(*

short summary
==================
This class tests all methods of LDT assertions
with various combinations of inputs and checks expected 
outputs are satisfied or not

.. <legal notes>

legal notes
=================
| SPDX-FileCopyrightText: © 2022 ekvip automation GmbH <info@ekvip.de>
| SPDX-License-Identifier: Apache-2.0
| For details check: Apache-2.0_

.. _Apache-2.0: https://www.apache.org/licenses/LICENSE-2.0

.. </legal notes>

methods and properties
======================

*)


FUNCTION_BLOCK LDTAssertionTests EXTENDS AbstractAssertorTest
VAR
	
END_VAR
VAR CONSTANT
	(* prefix to unify the test names *)
	TEST_NAME_PREFIX		:STRING := 'assert.dateAndTime.long.dateAndTime.';
	(* max value of a LWORD *)
	{attribute 'hide'}
	MAX_LWORD				:LWORD := 16#FFFF_FFFF_FFFF_FFFF;
	(* min value of a LWORD *)
	{attribute 'hide'}
	MIN_LWORD				:LWORD := 16#0000_0000_0000_0000;
	(* only the msb is set *)
	{attribute 'hide'}
	MSB_ONLY				:LWORD := 16#8000_0000_0000_0000;
	(* only the msb is set *)
	{attribute 'hide'}
	LSB_ONLY				:LWORD := 16#0000_0000_0000_0001;
	(* all bits set except the msb *)
	{attribute 'hide'}
	WITHOUT_MSB 			:LWORD := 16#7FFF_FFFF_FFFF_FFFF;
	(* for every nibble is the msb set only *)
	{attribute 'hide'}
	ALL_NIBBLE_MSB			:LWORD := 16#8888_8888_8888_8888;
	(* for every nibble is the msb unset only *)
	{attribute 'hide'}
	WITHOUT_NIBBLE_MSB		:LWORD := 16#7777_7777_7777_7777;
	(* for every nibble is the lsb set only *)
	{attribute 'hide'}
	ALL_NIBBLE_LSB			:LWORD := 16#1111_1111_1111_1111;
	(* every bit is set except the lsb *)
	{attribute 'hide'}
	LSB_IS_UNSET			:LWORD := 16#FFFF__FFFF_FFFF_FFFE;
	(* max vale of date and time *)
	LDT_MAX					:LDT := TO_LDT(MAX_LWORD);
	(* min vale of date and time *)
	LDT_MIN					:LDT := TO_LDT(MIN_LWORD);
	(* only the msb is set *)
	LDT_MSB_ONLY			:LDT := TO_LDT(MSB_ONLY);
	(* all bits set except the msb *)
	LDT_WITHOUT_MSB 		:LDT := TO_LDT(WITHOUT_MSB);
	(* for every nibble is the msb set only *)
	LDT_ALL_NIBBLE_MSB		:LDT := TO_LDT(ALL_NIBBLE_MSB);
	(* for every nibble is the msb unset only *)
	LDT_WITHOUT_NIBBLE_MSB	:LDT := TO_LDT(WITHOUT_NIBBLE_MSB);
	(* for every nibble is the lsb set only *)
	LDT_ALL_NIBBLE_LSB		:LDT := TO_LDT(ALL_NIBBLE_LSB);	
	(* every bit is set except the lsb *)
	LDT_LSB_IS_UNSET		:LDT := TO_LDT(LSB_IS_UNSET);
	(* only the msb is set *)
	LDT_LSB_ONLY			:LDT := TO_LDT(LSB_ONLY);
END_VAR

THIS^.runValueIsEqualToTests();
THIS^.runValueIsGreaterThanTests();
THIS^.runValueIsInRangeOfTests();
THIS^.runValueIsLessThanTests();
THIS^.runValueIsMaxTests();
THIS^.runValueIsMinTests();
THIS^.runValueIsNotEqualToTests();

(*

short summary
==================
This test method is a helper function to create a unified test name

.. <legal notes>

legal notes
=================
| SPDX-FileCopyrightText: © 2022 ekvip automation GmbH <info@ekvip.de>
| SPDX-License-Identifier: Apache-2.0
| For details check: Apache-2.0_

.. _Apache-2.0: https://www.apache.org/licenses/LICENSE-2.0

.. </legal notes>

parameters
==========

*)

METHOD PROTECTED getTestNameFor :Tc2_System.T_MaxString
VAR_INPUT
	(* name of the method to test, to create a unified test name *)
	nameOfMethodToTest	:Tc2_System.T_MaxString;
END_VAR
getTestNameFor := Tc2_Standard.CONCAT(THIS^.TEST_NAME_PREFIX, nameOfMethodToTest);
END_METHOD

(*

short summary
==================
This test method tests ``assert.dateAndTime.long.dateAndTime.valueIsEqualTo``
method of CNM_AssertionInterfaces library with various inputs

.. <legal notes>

legal notes
=================
| SPDX-FileCopyrightText: © 2022 ekvip automation GmbH <info@ekvip.de>
| SPDX-License-Identifier: Apache-2.0
| For details check: Apache-2.0_

.. _Apache-2.0: https://www.apache.org/licenses/LICENSE-2.0

.. </legal notes>

*)

METHOD runValueIsEqualToTests
RETURN (NOT TcUnit.TEST_ORDERED(THIS^.getTestNameFor('valueIsEqualTo')));

THIS^.testValueIsEqualTo(
	valueToTest := THIS^.LDT_MAX,
	expected := THIS^.LDT_MAX
);
THIS^.testValueIsEqualTo(
	valueToTest := THIS^.LDT_MIN,
	expected := THIS^.LDT_MIN
);
THIS^.testValueIsEqualTo(
	valueToTest := THIS^.LDT_MIN,
	expected := THIS^.LDT_MAX
);
THIS^.testValueIsEqualTo(
	valueToTest := THIS^.LDT_MAX,
	expected := THIS^.LDT_MIN
);
THIS^.testValueIsEqualTo(
	valueToTest := THIS^.LDT_ALL_NIBBLE_LSB,
	expected := THIS^.LDT_ALL_NIBBLE_LSB
);
THIS^.testValueIsEqualTo(
	valueToTest := THIS^.LDT_LSB_ONLY,
	expected := THIS^.LDT_MSB_ONLY
);
THIS^.testValueIsEqualTo(
	valueToTest := THIS^.LDT_MSB_ONLY,
	expected := THIS^.LDT_MSB_ONLY
);
THIS^.testValueIsEqualTo(
	valueToTest := THIS^.LDT_MSB_ONLY,
	expected := THIS^.LDT_LSB_ONLY
);

TcUnit.TEST_FINISHED();
END_METHOD

(*

short summary
==================
This test method tests ``assert.dateAndTime.long.dateAndTime.valueIsGreaterThan``
method of CNM_AssertionInterfaces library with various inputs

.. <legal notes>

legal notes
=================
| SPDX-FileCopyrightText: © 2022 ekvip automation GmbH <info@ekvip.de>
| SPDX-License-Identifier: Apache-2.0
| For details check: Apache-2.0_

.. _Apache-2.0: https://www.apache.org/licenses/LICENSE-2.0

.. </legal notes>

*)

METHOD runValueIsGreaterThanTests
RETURN (NOT TcUnit.TEST_ORDERED(THIS^.getTestNameFor('valueIsGreaterThan')));

THIS^.testValueIsGreaterThan(
	valueToTest := THIS^.LDT_MAX,
	lessValue := THIS^.LDT_MAX
);
THIS^.testValueIsGreaterThan(
	valueToTest := THIS^.LDT_MIN,
	lessValue := THIS^.LDT_MIN
);
THIS^.testValueIsGreaterThan(
	valueToTest := THIS^.LDT_MIN,
	lessValue := THIS^.LDT_MAX
);
THIS^.testValueIsGreaterThan(
	valueToTest := THIS^.LDT_MAX,
	lessValue := THIS^.LDT_MIN
);
THIS^.testValueIsGreaterThan(
	valueToTest := THIS^.LDT_ALL_NIBBLE_LSB,
	lessValue := THIS^.LDT_ALL_NIBBLE_LSB
);
THIS^.testValueIsGreaterThan(
	valueToTest := THIS^.LDT_ALL_NIBBLE_MSB,
	lessValue := THIS^.LDT_ALL_NIBBLE_LSB
);
THIS^.testValueIsGreaterThan(
	valueToTest := THIS^.LDT_ALL_NIBBLE_LSB,
	lessValue := THIS^.LDT_ALL_NIBBLE_MSB
);
THIS^.testValueIsGreaterThan(
	valueToTest := THIS^.LDT_LSB_ONLY,
	lessValue := THIS^.LDT_MSB_ONLY
);
THIS^.testValueIsGreaterThan(
	valueToTest := THIS^.LDT_MSB_ONLY,
	lessValue := THIS^.LDT_MSB_ONLY
);
THIS^.testValueIsGreaterThan(
	valueToTest := THIS^.LDT_MSB_ONLY,
	lessValue := THIS^.LDT_LSB_ONLY
);
THIS^.testValueIsGreaterThan(
	valueToTest := THIS^.LDT_LSB_IS_UNSET,
	lessValue := THIS^.LDT_MAX
);
THIS^.testValueIsGreaterThan(
	valueToTest := THIS^.LDT_MAX,
	lessValue := THIS^.LDT_LSB_IS_UNSET
);

TcUnit.TEST_FINISHED();
END_METHOD

(*

short summary
==================
This test method tests ``assert.dateAndTime.long.dateAndTime.valueIsInRangeOf``
method of CNM_AssertionInterfaces library with various inputs

.. <legal notes>

legal notes
=================
| SPDX-FileCopyrightText: © 2022 ekvip automation GmbH <info@ekvip.de>
| SPDX-License-Identifier: Apache-2.0
| For details check: Apache-2.0_

.. _Apache-2.0: https://www.apache.org/licenses/LICENSE-2.0

.. </legal notes>

*)

METHOD runValueIsInRangeOfTests
RETURN (NOT TcUnit.TEST_ORDERED(THIS^.getTestNameFor('valueIsInRangeOf')));

THIS^.testValueIsInRangeOf(
	lowerLimit := THIS^.LDT_MIN,
	valueToTest := THIS^.LDT_MAX,
	upperLimit	:= THIS^.LDT_MAX
);
THIS^.testValueIsInRangeOf(
	lowerLimit := THIS^.LDT_MIN,
	valueToTest := THIS^.LDT_MIN,
	upperLimit	:= THIS^.LDT_MAX
);
THIS^.testValueIsInRangeOf(
	lowerLimit := THIS^.LDT_MAX,
	valueToTest := THIS^.LDT_MAX,
	upperLimit	:= THIS^.LDT_MIN
);
THIS^.testValueIsInRangeOf(
	lowerLimit := THIS^.LDT_MAX,
	valueToTest := THIS^.LDT_MIN,
	upperLimit	:= THIS^.LDT_MIN
);
THIS^.testValueIsInRangeOf(
	lowerLimit := THIS^.LDT_LSB_IS_UNSET,
	valueToTest := THIS^.LDT_MIN,
	upperLimit	:= THIS^.LDT_MAX
);
THIS^.testValueIsInRangeOf(
	lowerLimit := THIS^.LDT_MIN,
	valueToTest := THIS^.LDT_LSB_IS_UNSET,
	upperLimit	:= THIS^.LDT_MAX
);
THIS^.testValueIsInRangeOf(
	lowerLimit := THIS^.LDT_LSB_IS_UNSET,
	valueToTest := THIS^.LDT_LSB_IS_UNSET,
	upperLimit	:= THIS^.LDT_LSB_IS_UNSET
);
THIS^.testValueIsInRangeOf(
	lowerLimit := THIS^.LDT_ALL_NIBBLE_LSB,
	valueToTest := THIS^.LDT_LSB_IS_UNSET,
	upperLimit	:= THIS^.LDT_ALL_NIBBLE_MSB
);
THIS^.testValueIsInRangeOf(
	lowerLimit := THIS^.LDT_LSB_IS_UNSET,
	valueToTest := THIS^.LDT_ALL_NIBBLE_LSB,
	upperLimit	:= THIS^.LDT_ALL_NIBBLE_MSB
);
THIS^.testValueIsInRangeOf(
	lowerLimit := THIS^.LDT_LSB_ONLY,
	valueToTest := THIS^.LDT_WITHOUT_MSB,
	upperLimit	:= THIS^.LDT_MSB_ONLY
);
THIS^.testValueIsInRangeOf(
	lowerLimit := THIS^.LDT_WITHOUT_MSB,
	valueToTest := THIS^.LDT_LSB_ONLY,
	upperLimit	:= THIS^.LDT_MSB_ONLY
);
THIS^.testValueIsInRangeOf(
	lowerLimit := THIS^.LDT_WITHOUT_NIBBLE_MSB,
	valueToTest := THIS^.LDT_MAX,
	upperLimit	:= THIS^.LDT_ALL_NIBBLE_MSB
);
THIS^.testValueIsInRangeOf(
	lowerLimit := THIS^.LDT_WITHOUT_NIBBLE_MSB,
	valueToTest := THIS^.LDT_MIN,
	upperLimit	:= THIS^.LDT_ALL_NIBBLE_MSB
);
THIS^.testValueIsInRangeOf(
	lowerLimit := THIS^.LDT_WITHOUT_NIBBLE_MSB,
	valueToTest := THIS^.LDT_WITHOUT_NIBBLE_MSB,
	upperLimit	:= THIS^.LDT_ALL_NIBBLE_MSB
);
THIS^.testValueIsInRangeOf(
	lowerLimit := THIS^.LDT_WITHOUT_NIBBLE_MSB,
	valueToTest := THIS^.LDT_ALL_NIBBLE_MSB,
	upperLimit	:= THIS^.LDT_ALL_NIBBLE_MSB
);

TcUnit.TEST_FINISHED();
END_METHOD

(*

short summary
==================
This test method tests ``assert.dateAndTime.long.dateAndTime.valueIsLessThan``
method of CNM_AssertionInterfaces library with various inputs

.. <legal notes>

legal notes
=================
| SPDX-FileCopyrightText: © 2022 ekvip automation GmbH <info@ekvip.de>
| SPDX-License-Identifier: Apache-2.0
| For details check: Apache-2.0_

.. _Apache-2.0: https://www.apache.org/licenses/LICENSE-2.0

.. </legal notes>

*)

METHOD runValueIsLessThanTests
RETURN (NOT TcUnit.TEST_ORDERED(THIS^.getTestNameFor('valueIsLessThan')));

THIS^.testValueIsLessThan(
	valueToTest := THIS^.LDT_MAX,
	greaterValue := THIS^.LDT_MAX
);
THIS^.testValueIsLessThan(
	valueToTest := THIS^.LDT_MIN,
	greaterValue := THIS^.LDT_MIN
);
THIS^.testValueIsLessThan(
	valueToTest := THIS^.LDT_MIN,
	greaterValue := THIS^.LDT_MAX
);
THIS^.testValueIsLessThan(
	valueToTest := THIS^.LDT_MAX,
	greaterValue := THIS^.LDT_MIN
);
THIS^.testValueIsLessThan(
	valueToTest := THIS^.LDT_ALL_NIBBLE_LSB,
	greaterValue := THIS^.LDT_ALL_NIBBLE_LSB
);
THIS^.testValueIsLessThan(
	valueToTest := THIS^.LDT_ALL_NIBBLE_MSB,
	greaterValue := THIS^.LDT_ALL_NIBBLE_LSB
);
THIS^.testValueIsLessThan(
	valueToTest := THIS^.LDT_ALL_NIBBLE_LSB,
	greaterValue := THIS^.LDT_ALL_NIBBLE_MSB
);
THIS^.testValueIsLessThan(
	valueToTest := THIS^.LDT_LSB_ONLY,
	greaterValue := THIS^.LDT_MSB_ONLY
);
THIS^.testValueIsLessThan(
	valueToTest := THIS^.LDT_MSB_ONLY,
	greaterValue := THIS^.LDT_MSB_ONLY
);
THIS^.testValueIsLessThan(
	valueToTest := THIS^.LDT_MSB_ONLY,
	greaterValue := THIS^.LDT_LSB_ONLY
);
THIS^.testValueIsLessThan(
	valueToTest := THIS^.LDT_LSB_IS_UNSET,
	greaterValue := THIS^.LDT_MAX
);
THIS^.testValueIsLessThan(
	valueToTest := THIS^.LDT_MAX,
	greaterValue := THIS^.LDT_LSB_IS_UNSET
);

TcUnit.TEST_FINISHED();
END_METHOD

(*

short summary
==================
This test method tests ``assert.dateAndTime.long.dateAndTime.valueIsMax``
method of CNM_AssertionInterfaces library with various inputs

.. <legal notes>

legal notes
=================
| SPDX-FileCopyrightText: © 2022 ekvip automation GmbH <info@ekvip.de>
| SPDX-License-Identifier: Apache-2.0
| For details check: Apache-2.0_

.. _Apache-2.0: https://www.apache.org/licenses/LICENSE-2.0

.. </legal notes>

*)

METHOD runValueIsMaxTests
RETURN (NOT TcUnit.TEST_ORDERED(THIS^.getTestNameFor('valueIsMax')));

THIS^.testValueIsMax(
	valueToTest := THIS^.LDT_MAX,
	maximumValue := THIS^.LDT_MAX
);
THIS^.testValueIsMax(
	valueToTest := THIS^.LDT_MIN,
	maximumValue := THIS^.LDT_MIN
);
THIS^.testValueIsMax(
	valueToTest := THIS^.LDT_MIN,
	maximumValue := THIS^.LDT_MAX
);
THIS^.testValueIsMax(
	valueToTest := THIS^.LDT_MAX,
	maximumValue := THIS^.LDT_MIN
);
THIS^.testValueIsMax(
	valueToTest := THIS^.LDT_ALL_NIBBLE_LSB,
	maximumValue := THIS^.LDT_ALL_NIBBLE_LSB
);
THIS^.testValueIsMax(
	valueToTest := THIS^.LDT_ALL_NIBBLE_MSB,
	maximumValue := THIS^.LDT_ALL_NIBBLE_LSB
);
THIS^.testValueIsMax(
	valueToTest := THIS^.LDT_ALL_NIBBLE_LSB,
	maximumValue := THIS^.LDT_ALL_NIBBLE_MSB
);
THIS^.testValueIsMax(
	valueToTest := THIS^.LDT_LSB_ONLY,
	maximumValue := THIS^.LDT_MSB_ONLY
);
THIS^.testValueIsMax(
	valueToTest := THIS^.LDT_MSB_ONLY,
	maximumValue := THIS^.LDT_MSB_ONLY
);
THIS^.testValueIsMax(
	valueToTest := THIS^.LDT_MSB_ONLY,
	maximumValue := THIS^.LDT_LSB_ONLY
);
THIS^.testValueIsMax(
	valueToTest := THIS^.LDT_LSB_IS_UNSET,
	maximumValue := THIS^.LDT_MAX
);
THIS^.testValueIsMax(
	valueToTest := THIS^.LDT_MAX,
	maximumValue := THIS^.LDT_LSB_IS_UNSET
);

TcUnit.TEST_FINISHED();
END_METHOD

(*

short summary
==================
This test method tests ``assert.dateAndTime.long.dateAndTime.valueIsMin``
method of CNM_AssertionInterfaces library with various inputs

.. <legal notes>

legal notes
=================
| SPDX-FileCopyrightText: © 2022 ekvip automation GmbH <info@ekvip.de>
| SPDX-License-Identifier: Apache-2.0
| For details check: Apache-2.0_

.. _Apache-2.0: https://www.apache.org/licenses/LICENSE-2.0

.. </legal notes>

*)

METHOD runValueIsMinTests
RETURN (NOT TcUnit.TEST_ORDERED(THIS^.getTestNameFor('valueIsMin')));

THIS^.testValueIsMin(
	valueToTest := THIS^.LDT_MAX,
	minimumValue := THIS^.LDT_MAX
);
THIS^.testValueIsMin(
	valueToTest := THIS^.LDT_MIN,
	minimumValue := THIS^.LDT_MIN
);
THIS^.testValueIsMin(
	valueToTest := THIS^.LDT_MIN,
	minimumValue := THIS^.LDT_MAX
);
THIS^.testValueIsMin(
	valueToTest := THIS^.LDT_MAX,
	minimumValue := THIS^.LDT_MIN
);
THIS^.testValueIsMin(
	valueToTest := THIS^.LDT_ALL_NIBBLE_LSB,
	minimumValue := THIS^.LDT_ALL_NIBBLE_LSB
);
THIS^.testValueIsMin(
	valueToTest := THIS^.LDT_ALL_NIBBLE_MSB,
	minimumValue := THIS^.LDT_ALL_NIBBLE_LSB
);
THIS^.testValueIsMin(
	valueToTest := THIS^.LDT_ALL_NIBBLE_LSB,
	minimumValue := THIS^.LDT_ALL_NIBBLE_MSB
);
THIS^.testValueIsMin(
	valueToTest := THIS^.LDT_LSB_ONLY,
	minimumValue := THIS^.LDT_MSB_ONLY
);
THIS^.testValueIsMin(
	valueToTest := THIS^.LDT_MSB_ONLY,
	minimumValue := THIS^.LDT_MSB_ONLY
);
THIS^.testValueIsMin(
	valueToTest := THIS^.LDT_MSB_ONLY,
	minimumValue := THIS^.LDT_LSB_ONLY
);
THIS^.testValueIsMin(
	valueToTest := THIS^.LDT_LSB_IS_UNSET,
	minimumValue := THIS^.LDT_MAX
);
THIS^.testValueIsMin(
	valueToTest := THIS^.LDT_MAX,
	minimumValue := THIS^.LDT_LSB_IS_UNSET
);

TcUnit.TEST_FINISHED();
END_METHOD

(*

short summary
==================
This test method tests ``assert.dateAndTime.long.dateAndTime.valueIsNotEqualTo``
method of CNM_AssertionInterfaces library with various inputs

.. <legal notes>

legal notes
=================
| SPDX-FileCopyrightText: © 2022 ekvip automation GmbH <info@ekvip.de>
| SPDX-License-Identifier: Apache-2.0
| For details check: Apache-2.0_

.. _Apache-2.0: https://www.apache.org/licenses/LICENSE-2.0

.. </legal notes>

*)

METHOD runValueIsNotEqualToTests
RETURN (NOT TcUnit.TEST_ORDERED(THIS^.getTestNameFor('valueIsNotEqualTo')));

THIS^.testValueIsNotEqualTo(
	valueToTest := THIS^.LDT_MAX,
	unexpectedValue := THIS^.LDT_MAX
);
THIS^.testValueIsNotEqualTo(
	valueToTest := THIS^.LDT_MIN,
	unexpectedValue := THIS^.LDT_MIN
);
THIS^.testValueIsNotEqualTo(
	valueToTest := THIS^.LDT_MIN,
	unexpectedValue := THIS^.LDT_MAX
);
THIS^.testValueIsNotEqualTo(
	valueToTest := THIS^.LDT_MAX,
	unexpectedValue := THIS^.LDT_MIN
);
THIS^.testValueIsNotEqualTo(
	valueToTest := THIS^.LDT_ALL_NIBBLE_LSB,
	unexpectedValue := THIS^.LDT_ALL_NIBBLE_LSB
);
THIS^.testValueIsNotEqualTo(
	valueToTest := THIS^.LDT_LSB_ONLY,
	unexpectedValue := THIS^.LDT_MSB_ONLY
);
THIS^.testValueIsNotEqualTo(
	valueToTest := THIS^.LDT_MSB_ONLY,
	unexpectedValue := THIS^.LDT_MSB_ONLY
);
THIS^.testValueIsNotEqualTo(
	valueToTest := THIS^.LDT_MSB_ONLY,
	unexpectedValue := THIS^.LDT_LSB_ONLY
);

TcUnit.TEST_FINISHED();
END_METHOD

(*

short summary
==================
This test method tests ``assert.dateAndTime.long.dateAndTime.valueIsEqualTo``
method of CNM_AssertionInterfaces library, 
it provides the possibility to handover test data via parameter 


.. <legal notes>

legal notes
=================
| SPDX-FileCopyrightText: © 2022 ekvip automation GmbH <info@ekvip.de>
| SPDX-License-Identifier: Apache-2.0
| For details check: Apache-2.0_

.. _Apache-2.0: https://www.apache.org/licenses/LICENSE-2.0

.. </legal notes>

parameters
==========

*)

METHOD testValueIsEqualTo 
VAR_INPUT
	(* for the test it's the parameter ``currentValue`` *)
	valueToTest	:LDT;
	(* for the test it's the parameter ``expectedValue`` *)
	expected	:LDT;
END_VAR
VAR
	(* just the expectation if the assertion to test must be worng or true *)
	assertionIsWrong		:BOOL;
	(* contains the format string for the test message *)
	message					:Tc2_System.T_MaxString;
	(* TwinCAT printf with the test message *)
	messageStringBuilder	:Tc2_Utilities.FB_FormatString;
	(* LDT value of ``currentValue`` as string *)
	currentValueAsString	:STRING(22);
	(* LDT value of ``expectedValue`` as string *)
	expectedValueAsString	:STRING(22);
END_VAR
THIS^.assertorContainer.resetAssertor();

assertionIsWrong := (valueToTest <> expected);

message := SEL(
	assertionIsWrong,
	'currentValue is %s expectedValue is %s assertion must be TRUE', 
	'currentValue is %s expectedValue is %s assertion must be FALSE'
);
currentValueAsString := TO_STRING(valueToTest);
expectedValueAsString := TO_STRING(expected);

messageStringBuilder(
	sFormat := message,
	arg1 := THIS^.AnyToArg(currentValueAsString),
	arg2 := THIS^.AnyToArg(expectedValueAsString)
);

THIS^.assertorContainer.assertor.assert.dateAndTime.long.dateAndTime.valueIsEqualTo(
	currentValue	:= valueToTest,
	expectedValue	:= expected,
	message			:= ''
);

THIS^.AssertEquals_BOOL(
	Expected 	:= assertionIsWrong,
	Actual 		:= THIS^.assertorContainer.wasAssertionWrong,
	Message 	:= messageStringBuilder.sOut
);
END_METHOD

(*

short summary
==================
This test method tests ``assert.dateAndTime.long.dateAndTime.valueIsGreaterThan``
method of CNM_AssertionInterfaces library, 
it provides the possibility to handover test data via parameter 


.. <legal notes>

legal notes
=================
| SPDX-FileCopyrightText: © 2022 ekvip automation GmbH <info@ekvip.de>
| SPDX-License-Identifier: Apache-2.0
| For details check: Apache-2.0_

.. _Apache-2.0: https://www.apache.org/licenses/LICENSE-2.0

.. </legal notes>

parameters
==========

*)

METHOD testValueIsGreaterThan 
VAR_INPUT
	(* for the test it's the parameter ``currentValue`` *)
	valueToTest	:LDT;
	(* for the test it's the parameter ``lessValue`` *)
	lessValue	:LDT;
END_VAR
VAR
	(* just the expectation if the assertion to test must be worng or true *)
	assertionIsWrong		:BOOL;
	(* contains the format string for the test message *)
	message					:Tc2_System.T_MaxString;
	(* TwinCAT printf with the test message *)
	messageStringBuilder	:Tc2_Utilities.FB_FormatString;
	(* LDT value of ``currentValue`` as string *)
	currentValueAsString	:STRING(22);
	(* LDT value of ``lessValue`` as string *)
	lessValueAsString		:STRING(22);
END_VAR
THIS^.assertorContainer.resetAssertor();

assertionIsWrong := (valueToTest <= lessValue);

message := SEL(
	assertionIsWrong,
	'currentValue is %s lessValue is %s assertion must be TRUE', 
	'currentValue is %s lessValue is %s assertion must be FALSE'
);
currentValueAsString := TO_STRING(valueToTest);
lessValueAsString := TO_STRING(lessValue);

messageStringBuilder(
	sFormat := message,
	arg1 := THIS^.AnyToArg(currentValueAsString),
	arg2 := THIS^.AnyToArg(lessValueAsString)
);

THIS^.assertorContainer.assertor.assert.dateAndTime.long.dateAndTime.valueIsGreaterThan(
	currentValue	:= valueToTest,
	lessValue		:= lessValue,
	message			:= ''
);

THIS^.AssertEquals_BOOL(
	Expected 	:= assertionIsWrong,
	Actual 		:= THIS^.assertorContainer.wasAssertionWrong,
	Message 	:= messageStringBuilder.sOut
);
END_METHOD

(*

short summary
==================
This test method tests ``assert.dateAndTime.long.dateAndTime.valueIsInRangeOf``
method of CNM_AssertionInterfaces library, 
it provides the possibility to handover test data via parameter 


.. <legal notes>

legal notes
=================
| SPDX-FileCopyrightText: © 2022 ekvip automation GmbH <info@ekvip.de>
| SPDX-License-Identifier: Apache-2.0
| For details check: Apache-2.0_

.. _Apache-2.0: https://www.apache.org/licenses/LICENSE-2.0

.. </legal notes>

parameters
==========

*)

METHOD testValueIsInRangeOf 
VAR_INPUT
	(* for the test it's the parameter ``lowerLimit`` *)
	lowerLimit	:LDT;
	(* for the test it's the parameter ``currentValue`` *)
	valueToTest	:LDT;
	(* for the test it's the parameter ``upperLimit`` *)
	upperLimit	:LDT;
END_VAR
VAR
	(* just the expectation if the assertion to test must be worng or true *)
	assertionIsWrong		:BOOL;
	(* contains the format string for the test message *)
	message					:Tc2_System.T_MaxString;
	(* TwinCAT printf with the test message *)
	messageStringBuilder	:Tc2_Utilities.FB_FormatString;
	(* LDT value of ``lowerLimit`` as string *)
	lowerLimitAsString		:STRING(22);
	(* LDT value of ``currentValue`` as string *)
	currentValueAsString	:STRING(22);
	(* dt value of ``upperLimit`` as string *)
	upperLimitAsString		:STRING(22);

END_VAR
THIS^.assertorContainer.resetAssertor();

assertionIsWrong := ((
		valueToTest < lowerLimit
	) OR (
		valueToTest > upperLimit
	)
);

message := SEL(
	assertionIsWrong,
	'lowerLimit is %s currentValue is %s upperLimit is %s assertion must be TRUE', 
	'lowerLimit is %s currentValue is %s upperLimit is %s assertion must be FALSE'
);
lowerLimitAsString		:= TO_STRING(lowerLimit);
currentValueAsString	:= TO_STRING(valueToTest);
upperLimitAsString		:= TO_STRING(upperLimit);

messageStringBuilder(
	sFormat := message,
	arg1 := THIS^.AnyToArg(lowerLimitAsString),
	arg2 := THIS^.AnyToArg(currentValueAsString),
	arg3 := THIS^.AnyToArg(upperLimitAsString)
);

THIS^.assertorContainer.assertor.assert.dateAndTime.long.dateAndTime.valueIsInRangeOf(
	lowerLimit		:= lowerLimit,
	currentValue	:= valueToTest,
	upperLimit		:= upperLimit,
	message			:= ''
);

THIS^.AssertEquals_BOOL(
	Expected 	:= assertionIsWrong,
	Actual 		:= THIS^.assertorContainer.wasAssertionWrong,
	Message 	:= messageStringBuilder.sOut
);
END_METHOD

(*

short summary
==================
This test method tests ``assert.dateAndTime.long.dateAndTime.valueIsLessThan``
method of CNM_AssertionInterfaces library, 
it provides the possibility to handover test data via parameter 


.. <legal notes>

legal notes
=================
| SPDX-FileCopyrightText: © 2022 ekvip automation GmbH <info@ekvip.de>
| SPDX-License-Identifier: Apache-2.0
| For details check: Apache-2.0_

.. _Apache-2.0: https://www.apache.org/licenses/LICENSE-2.0

.. </legal notes>

parameters
==========

*)

METHOD testValueIsLessThan 
VAR_INPUT
	(* for the test it's the parameter ``currentValue`` *)
	valueToTest		:LDT;
	(* for the test it's the parameter ``greaterValue`` *)
	greaterValue	:LDT;
END_VAR
VAR
	(* just the expectation if the assertion to test must be worng or true *)
	assertionIsWrong		:BOOL;
	(* contains the format string for the test message *)
	message					:Tc2_System.T_MaxString;
	(* TwinCAT printf with the test message *)
	messageStringBuilder	:Tc2_Utilities.FB_FormatString;
	(* LDT value of ``currentValue`` as string *)
	currentValueAsString	:STRING(22);
	(* LDT value of ``greaterValue`` as string *)
	greaterValueAsString	:STRING(22);
END_VAR
THIS^.assertorContainer.resetAssertor();

assertionIsWrong := (valueToTest >= greaterValue);

message := SEL(
	assertionIsWrong,
	'currentValue is %s greaterValue is %s assertion must be TRUE', 
	'currentValue is %s greaterValue is %s assertion must be FALSE'
);
currentValueAsString := TO_STRING(valueToTest);
greaterValueAsString := TO_STRING(greaterValue);

messageStringBuilder(
	sFormat := message,
	arg1 := THIS^.AnyToArg(currentValueAsString),
	arg2 := THIS^.AnyToArg(greaterValueAsString)
);

THIS^.assertorContainer.assertor.assert.dateAndTime.long.dateAndTime.valueIsLessThan(
	currentValue	:= valueToTest,
	greaterValue	:= greaterValue,
	message			:= ''
);

THIS^.AssertEquals_BOOL(
	Expected 	:= assertionIsWrong,
	Actual 		:= THIS^.assertorContainer.wasAssertionWrong,
	Message 	:= messageStringBuilder.sOut
);
END_METHOD

(*

short summary
==================
This test method tests ``assert.dateAndTime.long.dateAndTime.valueIsMax``
method of CNM_AssertionInterfaces library, 
it provides the possibility to handover test data via parameter 


.. <legal notes>

legal notes
=================
| SPDX-FileCopyrightText: © 2022 ekvip automation GmbH <info@ekvip.de>
| SPDX-License-Identifier: Apache-2.0
| For details check: Apache-2.0_

.. _Apache-2.0: https://www.apache.org/licenses/LICENSE-2.0

.. </legal notes>

parameters
==========

*)

METHOD testValueIsMax 
VAR_INPUT
	(* for the test it's the parameter ``currentValue`` *)
	valueToTest		:LDT;
	(* for the test it's the parameter ``greaterValue`` *)
	maximumValue	:LDT;
END_VAR
VAR
	(* just the expectation if the assertion to test must be worng or true *)
	assertionIsWrong		:BOOL;
	(* contains the format string for the test message *)
	message					:Tc2_System.T_MaxString;
	(* TwinCAT printf with the test message *)
	messageStringBuilder	:Tc2_Utilities.FB_FormatString;
	(* LDT value of ``currentValue`` as string *)
	currentValueAsString	:STRING(22);
	(* LDT value of ``maximumValue`` as string *)
	maximumValueAsString	:STRING(22);
END_VAR
THIS^.assertorContainer.resetAssertor();

assertionIsWrong := (valueToTest > maximumValue);

message := SEL(
	assertionIsWrong,
	'currentValue is %s maximumValue is %s assertion must be TRUE', 
	'currentValue is %s maximumValue is %s assertion must be FALSE'
);
currentValueAsString := TO_STRING(valueToTest);
maximumValueAsString := TO_STRING(maximumValue);

messageStringBuilder(
	sFormat := message,
	arg1 := THIS^.AnyToArg(currentValueAsString),
	arg2 := THIS^.AnyToArg(maximumValueAsString)
);

THIS^.assertorContainer.assertor.assert.dateAndTime.long.dateAndTime.valueIsMax(
	currentValue	:= valueToTest,
	maximumValue	:= maximumValue,
	message			:= ''
);

THIS^.AssertEquals_BOOL(
	Expected 	:= assertionIsWrong,
	Actual 		:= THIS^.assertorContainer.wasAssertionWrong,
	Message 	:= messageStringBuilder.sOut
);
END_METHOD

(*

short summary
==================
This test method tests ``assert.dateAndTime.long.dateAndTime.valueIsMin``
method of CNM_AssertionInterfaces library, 
it provides the possibility to handover test data via parameter 


.. <legal notes>

legal notes
=================
| SPDX-FileCopyrightText: © 2022 ekvip automation GmbH <info@ekvip.de>
| SPDX-License-Identifier: Apache-2.0
| For details check: Apache-2.0_

.. _Apache-2.0: https://www.apache.org/licenses/LICENSE-2.0

.. </legal notes>

parameters
==========

*)

METHOD testValueIsMin 
VAR_INPUT
	(* for the test it's the parameter ``currentValue`` *)
	valueToTest		:LDT;
	(* for the test it's the parameter ``greaterValue`` *)
	minimumValue	:LDT;
END_VAR
VAR
	(* just the expectation if the assertion to test must be worng or true *)
	assertionIsWrong		:BOOL;
	(* contains the format string for the test message *)
	message					:Tc2_System.T_MaxString;
	(* TwinCAT printf with the test message *)
	messageStringBuilder	:Tc2_Utilities.FB_FormatString;
	(* LDT value of ``currentValue`` as string *)
	currentValueAsString	:STRING(22);
	(* LDT value of ``minimumValue`` as string *)
	minimumValueAsString	:STRING(22);
END_VAR
THIS^.assertorContainer.resetAssertor();

assertionIsWrong := (valueToTest < minimumValue);

message := SEL(
	assertionIsWrong,
	'currentValue is %s minimumValue is %s assertion must be TRUE', 
	'currentValue is %s minimumValue is %s assertion must be FALSE'
);
currentValueAsString := TO_STRING(valueToTest);
minimumValueAsString := TO_STRING(minimumValue);

messageStringBuilder(
	sFormat := message,
	arg1 := THIS^.AnyToArg(currentValueAsString),
	arg2 := THIS^.AnyToArg(minimumValueAsString)
);

THIS^.assertorContainer.assertor.assert.dateAndTime.long.dateAndTime.valueIsMin(
	currentValue	:= valueToTest,
	minimumValue	:= minimumValue,
	message			:= ''
);

THIS^.AssertEquals_BOOL(
	Expected 	:= assertionIsWrong,
	Actual 		:= THIS^.assertorContainer.wasAssertionWrong,
	Message 	:= messageStringBuilder.sOut
);
END_METHOD

(*

short summary
==================
This test method tests ``assert.dateAndTime.long.dateAndTime.valueIsNotEqualTo``
method of CNM_AssertionInterfaces library, 
it provides the possibility to handover test data via parameter 


.. <legal notes>

legal notes
=================
| SPDX-FileCopyrightText: © 2022 ekvip automation GmbH <info@ekvip.de>
| SPDX-License-Identifier: Apache-2.0
| For details check: Apache-2.0_

.. _Apache-2.0: https://www.apache.org/licenses/LICENSE-2.0

.. </legal notes>

parameters
==========

*)

METHOD testValueIsNotEqualTo 
VAR_INPUT
	(* for the test it's the parameter ``currentValue`` *)
	valueToTest		:LDT;
	(* for the test it's the parameter ``unexpectedValue`` *)
	unexpectedValue	:LDT;
END_VAR
VAR
	(* just the expectation if the assertion to test must be worng or true *)
	assertionIsWrong		:BOOL;
	(* contains the format string for the test message *)
	message					:Tc2_System.T_MaxString;
	(* TwinCAT printf with the test message *)
	messageStringBuilder	:Tc2_Utilities.FB_FormatString;
	(* LDT value of ``currentValue`` as string *)
	currentValueAsString	:STRING(22);
	(* LDT value of ``unexpectedValue`` as string *)
	unexpectedValueAsString	:STRING(22);
END_VAR
THIS^.assertorContainer.resetAssertor();

assertionIsWrong := (valueToTest = unexpectedValue);

message := SEL(
	assertionIsWrong,
	'currentValue is %s expectedValue is %s assertion must be TRUE', 
	'currentValue is %s expectedValue is %s assertion must be FALSE'
);
currentValueAsString := TO_STRING(valueToTest);
unexpectedValueAsString := TO_STRING(unexpectedValue);

messageStringBuilder(
	sFormat := message,
	arg1 := THIS^.AnyToArg(currentValueAsString),
	arg2 := THIS^.AnyToArg(unexpectedValueAsString)
);

THIS^.assertorContainer.assertor.assert.dateAndTime.long.dateAndTime.valueIsNotEqualTo(
	currentValue	:= valueToTest,
	unexpectedValue	:= unexpectedValue,
	message			:= ''
);

THIS^.AssertEquals_BOOL(
	Expected 	:= assertionIsWrong,
	Actual 		:= THIS^.assertorContainer.wasAssertionWrong,
	Message 	:= messageStringBuilder.sOut
);
END_METHOD

END_FUNCTION_BLOCK

(* stored: Version 1.1.0.1, ProductVersion 3.1.4026.13
   POU LDTAssertionTests: Id {6a7ec885-b5af-4274-99d4-0f2e9afa3519}, SpecialFunc None
   Folder internal: Id {004530f2-5ef1-4ce5-a905-e6f6d0b90d24}
   Folder valueIsEqualTo: Id {8ac71dcc-1f22-4104-9799-d3e0d229ef01}
   Folder valueIsGreaterThan: Id {85a35603-cadb-4c36-9940-3dbfd893e8c2}
   Folder valueIsInRangeOf: Id {c30c595e-cb71-4a4f-8a5c-2202be460c45}
   Folder valueIsLessThan: Id {5043e7d3-afd0-4cb9-b4a0-93e5e37d7969}
   Folder valueIsMax: Id {ed632205-42df-42a9-9500-d9fa6c2ccbc7}
   Folder valueIsMin: Id {5632adcc-8ae7-4c74-a0bc-65ca43c1f2a2}
   Folder valueIsNotEqualTo: Id {808c3772-1ee8-4ef0-a6a2-9bc348b3c609}
   Method getTestNameFor: Id {c7c58e24-99c2-4974-ae36-65037fba4c7c}
   Method runValueIsEqualToTests: Id {d796edf3-7dad-47c3-835c-c0f9dd5e4cd0}
   Method runValueIsGreaterThanTests: Id {064d15db-12d4-4fd2-bda8-21839bb38c4f}
   Method runValueIsInRangeOfTests: Id {723fee2f-fbfe-4509-a99f-c49ecf80aae3}
   Method runValueIsLessThanTests: Id {df84ffc0-3bd4-4b14-94ce-c9fd8c8180eb}
   Method runValueIsMaxTests: Id {e49ed82c-99d8-474a-abdc-b7e6adbaefd2}
   Method runValueIsMinTests: Id {e622140d-d127-4463-8bec-9f316bfadd63}
   Method runValueIsNotEqualToTests: Id {da2979bf-3c9f-4c72-b277-815ea282bb9d}
   Method testValueIsEqualTo: Id {166601af-84df-44dc-9132-d5938279574f}
   Method testValueIsGreaterThan: Id {4a58a302-b6b7-40b8-a98e-adf1572e01a9}
   Method testValueIsInRangeOf: Id {d78ac551-3b7d-4ead-8416-e0f17be681d2}
   Method testValueIsLessThan: Id {66b94df4-22ed-4a84-b3cc-be6e2769abc7}
   Method testValueIsMax: Id {50ee1975-cb20-40ce-88f3-aac11b295b9d}
   Method testValueIsMin: Id {92b86a7f-81e9-43d7-8b70-bd5e82b243ae}
   Method testValueIsNotEqualTo: Id {a6e61558-de57-4add-8d75-fc9ce0f86c74} *)
